// TIA Portal V17 export
// export: Created 2025-03-05T08:02:17.9836067Z, ExportSetting WithDefaults, DisplayName Totally Integrated Automation Portal, DisplayVersion V17 Update 8, DisplayName TIA Portal Openness, DisplayVersion V17 Update 8, DisplayName TIA Portal Version Control Interface, DisplayVersion V17, DisplayName SINAMICS Startdrive Advanced, DisplayVersion V17 SP2, DisplayName SINAMICS Startdrive G110M, G120, G120C, G120D, G120P, G115D, DisplayVersion V17 SP2, DisplayName SINAMICS Startdrive G130, G150, S120, S150, SINAMICS MV, S210, DisplayVersion V17 SP2, DisplayName STEP 7 Professional, DisplayVersion V17 Update 8, DisplayName SINUMERIK ONE STEP 7 Toolbox, DisplayVersion V17 Update 12, DisplayName SINUMERIK 840D sl STEP 7 Toolbox, DisplayVersion V17 Update 12, DisplayName STEP 7 Safety, DisplayVersion V17 Update 6, DisplayName WinCC Advanced, DisplayVersion V17 Update 8
TYPE "HT10_INPUTS"
// stored: IsFailsafeCompliant false
   STRUCT
      SPARE_0_0 : Bool;   // SPARE 0 0
      RESET_FAULT_I : Bool;   // HT10 RESET FAULT INPUT
      SPARE_0_2 : Bool;   // SPARE 0 2
      SPARE_0_3 : Bool;   // SPARE 0 3
      SPARE_0_4 : Bool;   // SPARE 0 4
      SPARE_0_5 : Bool;   // SPARE 0 5
      SPARE_0_6 : Bool;   // SPARE 0 6
      SPARE_0_7 : Bool;   // SPARE 0 7
      SPARE_1_0 : Bool;   // SPARE 1 0
      SPARE_1_1 : Bool;   // SPARE 1 1
      U1 : Bool;   // SELECT MANUAL MODE
      U2 : Bool;   // SELECT REFERENCE MODE
      SPARE_1_4 : Bool;   // SPARE 1 4
      U3 : Bool;   // SELECT SEMIAUTO MODE
      U4 : Bool;   // SPARE 1 6
      U_OPTION_I : Bool;   // HT10 U OPTION INPUT
      SPARE_2 : Byte;   // SPARE 2
      SPARE_3_0 : Bool;   // SPARE 3 0
      SPARE_3_1 : Bool;   // SPARE 3 1
      SPARE_3_2 : Bool;   // SPARE 3 2
      SPARE_3_3 : Bool;   // SPARE 3 3
      SPARE_3_4 : Bool;   // SPARE 3 4
      SPARE_3_5 : Bool;   // SPARE 3 5
      JOG_MIINUS_I : Bool;   // HT10 JOG MIINUS INPUT
      JOG_PLUS_I : Bool;   // HT10 JOG PLUS INPUT
      U16 : Bool;   // SPARE 3 0
      U15 : Bool;   // SPARE 3 1
      U14 : Bool;   // SPARE 3 2
      U13 : Bool;   // SPARE 3 3
      U12 : Bool;   // SPARE 3 4
      U11 : Bool;   // SPARE 3 5
      U10 : Bool;   // SPARE 3 5
      U9 : Bool;   // SPARE 3 5
      RAPID_I : Bool;   // HT10 RAPID INPUT
      SPARE_5_1 : Bool;   // SPARE 5 1
      SPARE_5_2 : Bool;   // SPARE 5 2
      U5 : Bool;   // SPARE 5 3
      U6 : Bool;   // SPARE 5 4
      U7 : Bool;   // SPARE 5 5
      U8 : Bool;   // SPARE 5 6
      SPARE_5_7 : Bool;   // SPARE 5 7
      NC_STOP_I : Bool;   // HT10 NC STOP INPUT
      NC_START_I : Bool;   // HT10 NC START INPUT
      OVERRIDE_I : Byte;   // HT10 OVERRIDE INPUT
   END_STRUCT;
END_TYPE
